(* LS Electric XG5000 project: 10_Practice3_HMI_Control_Timer *)
(* PLC LSPLC *)

PROGRAM NewProgram (* task: 스캔 프로그램 *)
VAR
    OFF AT %IX0.0.1 : BOOL;
    ON AT %IX0.0.0 : BOOL;
    램프 AT %QX0.1.0 : BOOL;
    비트메세지 AT %MX0 : BOOL;
    시간입력 AT %MD0 : TIME := T#5s;
    시간출력 AT %MD10 : TIME;
    온타이머1 : TON;
END_VAR

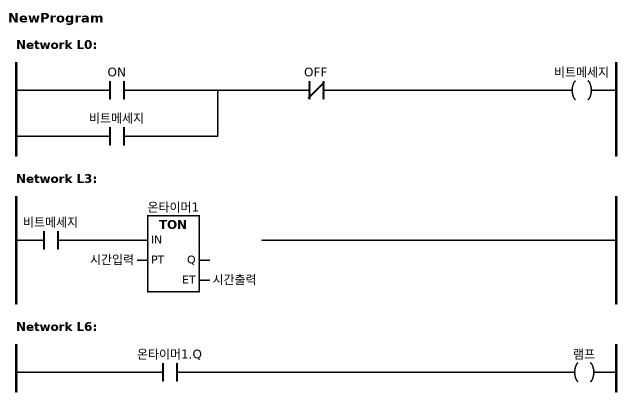
(* Rung L0 *)
비트메세지 := (ON OR 비트메세지) AND NOT OFF;
(* Rung L3 *)
온타이머1(IN := 비트메세지, PT := 시간입력, ET => 시간출력);
(* Rung L6 *)
램프 := 온타이머1.Q;
END_PROGRAM